Staubli VAL3: BackupProduct.pgx

public program BackupProduct(string x_sSFileName (dimensions=1), num x_nIndex (dimensions=1), bool x_b2Txt (dimensions=1))
begin
  call FileDir:CloseAllFile()

  //2013.10.30
  //一个工位可以选择多个产品，主要是为了法利莱
  if bMoreProd1Wp
    if $fileExists(x_sSFileName)
      if !$copy(x_sSFileName,"Disk://Txt/Product"+toString("",x_nIndex)+".txt")
        popUpMsg("复制文件出错")
        logMsg("复制文件出错")
      endIf
    endIf
    return
  endIf


  if x_b2Txt
    if $fileExists("Disk://BackUp/"+toString("",x_nIndex)+".txt")
      if !$copy("Disk://BackUp/"+toString("",x_nIndex)+".txt","Disk://Txt/product"+toString("",x_nIndex)+".txt")
        popUpMsg("复制文件出错")
      endIf
    endIf
  else
    if $fileExists(x_sSFileName)
      if !$copy(x_sSFileName,"Disk://BackUp/"+toString("",x_nIndex)+".txt")
        popUpMsg("复制文件出错")
      endIf
    endIf

  endIf















end
